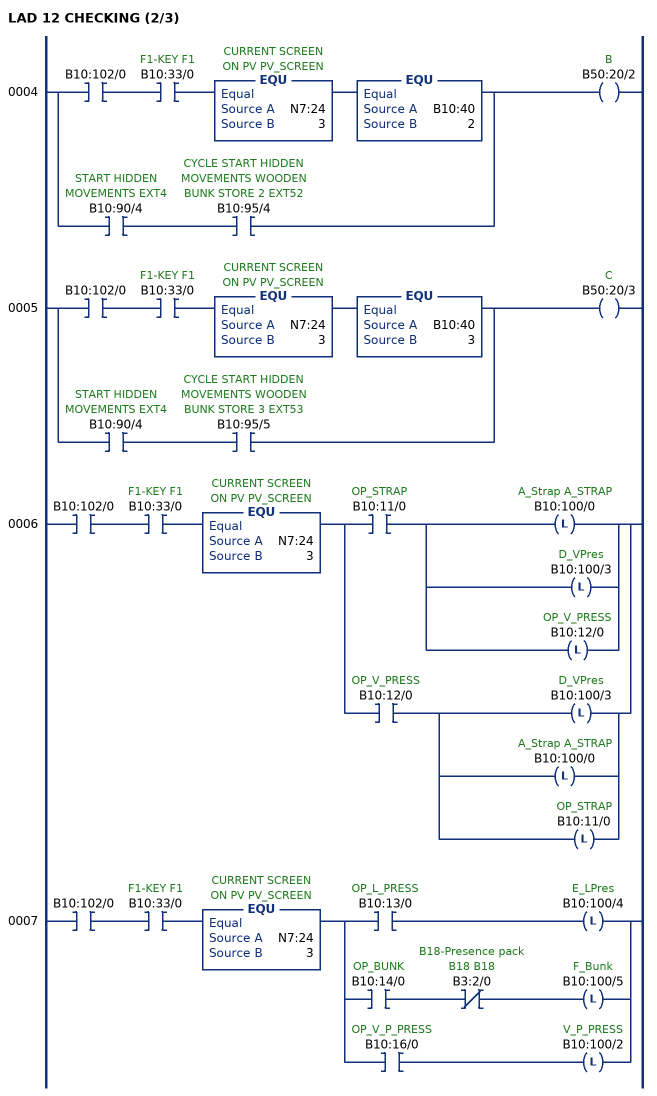
% Rung: 4 %
SOR BST XIC B10:102/0 XIC B10:33/0 EQU N7:24 3 EQU B10:40 2 NXB XIC B10:90/4 XIC B10:95/4 BND OTE B50:20/2 EOR
%   B10:33/0  F1  "F1-KEY" %
%   N7:24  PV_SCREEN  "CURRENT SCREEN ON PV" %
%   B10:90/4  EXT4  "START HIDDEN MOVEMENTS" %
%   B10:95/4  EXT52  "CYCLE START HIDDEN MOVEMENTS WOODEN BUNK STORE 2" %
%   B50:20/2  "B" %
% Rung: 5 %
SOR BST XIC B10:102/0 XIC B10:33/0 EQU N7:24 3 EQU B10:40 3 NXB XIC B10:90/4 XIC B10:95/5 BND OTE B50:20/3 EOR
%   B10:33/0  F1  "F1-KEY" %
%   N7:24  PV_SCREEN  "CURRENT SCREEN ON PV" %
%   B10:90/4  EXT4  "START HIDDEN MOVEMENTS" %
%   B10:95/5  EXT53  "CYCLE START HIDDEN MOVEMENTS WOODEN BUNK STORE 3" %
%   B50:20/3  "C" %
% Rung: 6 %
SOR XIC B10:102/0 XIC B10:33/0 EQU N7:24 3 BST XIC B10:11/0 BST OTL B10:100/0 NXB BST OTL B10:100/3 NXB OTL B10:12/0 BND BND NXB XIC B10:12/0 BST OTL B10:100/3 NXB BST OTL B10:100/0 NXB OTL B10:11/0 BND BND BND EOR
%   B10:33/0  F1  "F1-KEY" %
%   N7:24  PV_SCREEN  "CURRENT SCREEN ON PV" %
%   B10:11/0  "OP_STRAP" %
%   B10:100/0  A_STRAP  "A_Strap" %
%   B10:100/3  "D_VPres" %
%   B10:12/0  "OP_V_PRESS" %
% Rung: 7 %
SOR XIC B10:102/0 XIC B10:33/0 EQU N7:24 3 BST XIC B10:13/0 OTL B10:100/4 NXB BST XIC B10:14/0 XIO B3:2/0 OTL B10:100/5 NXB XIC B10:16/0 OTL B10:100/2 BND BND EOR
%   B10:33/0  F1  "F1-KEY" %
%   N7:24  PV_SCREEN  "CURRENT SCREEN ON PV" %
%   B10:13/0  "OP_L_PRESS" %
%   B10:100/4  "E_LPres" %
%   B10:14/0  "OP_BUNK" %
%   B3:2/0  B18  "B18-Presence pack B18" %
%   B10:100/5  "F_Bunk" %
%   B10:16/0  "OP_V_P_PRESS" %
%   B10:100/2  "V_P_PRESS" %

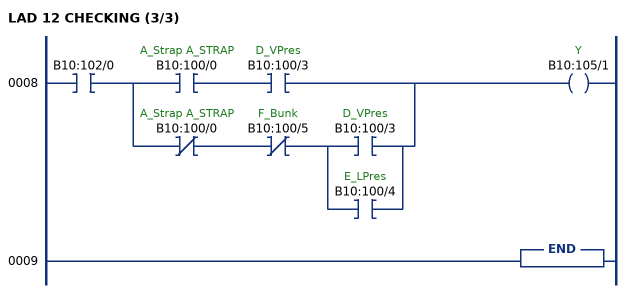
% Rung: 8 %
SOR XIC B10:102/0 BST XIC B10:100/0 XIC B10:100/3 NXB XIO B10:100/0 XIO B10:100/5 BST XIC B10:100/3 NXB XIC B10:100/4 BND BND OTE B10:105/1 EOR
%   B10:100/0  A_STRAP  "A_Strap" %
%   B10:100/3  "D_VPres" %
%   B10:100/5  "F_Bunk" %
%   B10:100/4  "E_LPres" %
%   B10:105/1  "Y" %
% Rung: 9 %
SOR END EOR

LADDER 13 "INFEED"    % INFEED CONTROLS %
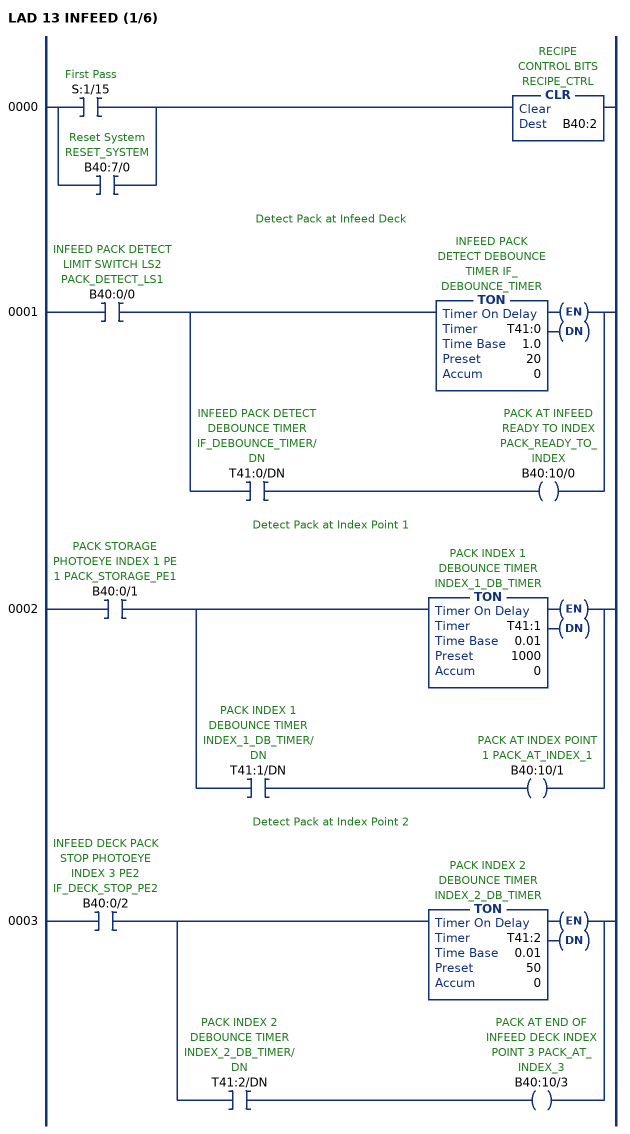
% Rung: 0 %
SOR BST XIC S:1/15 NXB XIC B40:7/0 BND CLR B40:2 EOR
%   S:1/15  "First Pass" %
%   B40:7/0  RESET_SYSTEM  "Reset System" %
%   B40:2  RECIPE_CTRL  "RECIPE CONTROL BITS" %
% Rung: 1 %
% Detect Pack at Infeed Deck %
SOR XIC B40:0/0 BST TON T41:0 1.0 20 0 NXB XIC T41:0/DN OTE B40:10/0 BND EOR
%   B40:0/0  PACK_DETECT_LS1  "INFEED PACK DETECT LIMIT SWITCH LS2" %
%   T41:0  IF_DEBOUNCE_TIMER  "INFEED PACK DETECT DEBOUNCE TIMER" %
%   B40:10/0  PACK_READY_TO_INDEX  "PACK AT INFEED READY TO INDEX" %
% Rung: 2 %
% Detect Pack at Index Point 1 %
SOR XIC B40:0/1 BST TON T41:1 0.01 1000 0 NXB XIC T41:1/DN OTE B40:10/1 BND EOR
%   B40:0/1  PACK_STORAGE_PE1  "PACK STORAGE PHOTOEYE INDEX 1 PE 1" %
%   T41:1  INDEX_1_DB_TIMER  "PACK INDEX 1 DEBOUNCE TIMER" %
%   B40:10/1  PACK_AT_INDEX_1  "PACK AT INDEX POINT 1" %
% Rung: 3 %
% Detect Pack at Index Point 2 %
SOR XIC B40:0/2 BST TON T41:2 0.01 50 0 NXB XIC T41:2/DN OTE B40:10/3 BND EOR
%   B40:0/2  IF_DECK_STOP_PE2  "INFEED DECK PACK STOP PHOTOEYE INDEX 3 PE2" %
%   T41:2  INDEX_2_DB_TIMER  "PACK INDEX 2 DEBOUNCE TIMER" %
%   B40:10/3  PACK_AT_INDEX_3  "PACK AT END OF INFEED DECK INDEX POINT 3" %

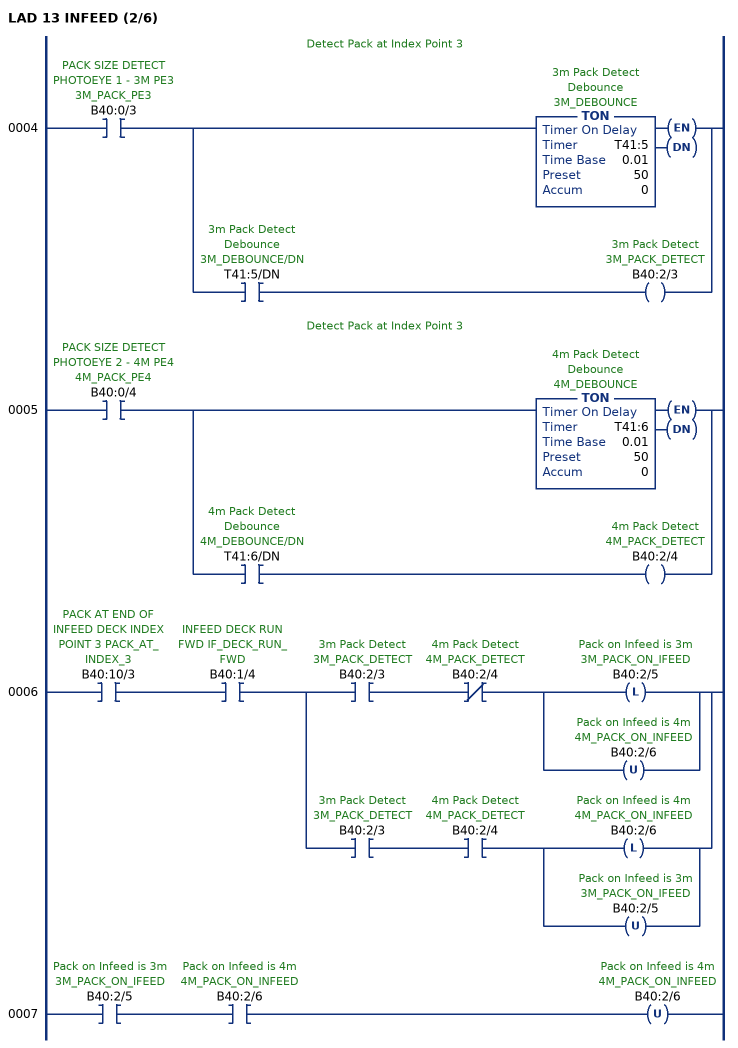
% Rung: 4 %
% Detect Pack at Index Point 3 %
SOR XIC B40:0/3 BST TON T41:5 0.01 50 0 NXB XIC T41:5/DN OTE B40:2/3 BND EOR
%   B40:0/3  3M_PACK_PE3  "PACK SIZE DETECT PHOTOEYE 1 - 3M PE3" %
%   T41:5  3M_DEBOUNCE  "3m Pack Detect Debounce" %
%   B40:2/3  3M_PACK_DETECT  "3m Pack Detect" %
% Rung: 5 %
% Detect Pack at Index Point 3 %
SOR XIC B40:0/4 BST TON T41:6 0.01 50 0 NXB XIC T41:6/DN OTE B40:2/4 BND EOR
%   B40:0/4  4M_PACK_PE4  "PACK SIZE DETECT PHOTOEYE 2 - 4M PE4" %
%   T41:6  4M_DEBOUNCE  "4m Pack Detect Debounce" %
%   B40:2/4  4M_PACK_DETECT  "4m Pack Detect" %
% Rung: 6 %
SOR XIC B40:10/3 XIC B40:1/4 BST XIC B40:2/3 XIO B40:2/4 BST OTL B40:2/5 NXB OTU B40:2/6 BND NXB XIC B40:2/3 XIC B40:2/4 BST OTL B40:2/6 NXB OTU B40:2/5 BND BND EOR
%   B40:10/3  PACK_AT_INDEX_3  "PACK AT END OF INFEED DECK INDEX POINT 3" %
%   B40:1/4  IF_DECK_RUN_FWD  "INFEED DECK RUN FWD" %
%   B40:2/3  3M_PACK_DETECT  "3m Pack Detect" %
%   B40:2/4  4M_PACK_DETECT  "4m Pack Detect" %
%   B40:2/5  3M_PACK_ON_IFEED  "Pack on Infeed is 3m" %
%   B40:2/6  4M_PACK_ON_INFEED  "Pack on Infeed is 4m" %
% Rung: 7 %
SOR XIC B40:2/5 XIC B40:2/6 OTU B40:2/6 EOR
%   B40:2/5  3M_PACK_ON_IFEED  "Pack on Infeed is 3m" %
%   B40:2/6  4M_PACK_ON_INFEED  "Pack on Infeed is 4m" %

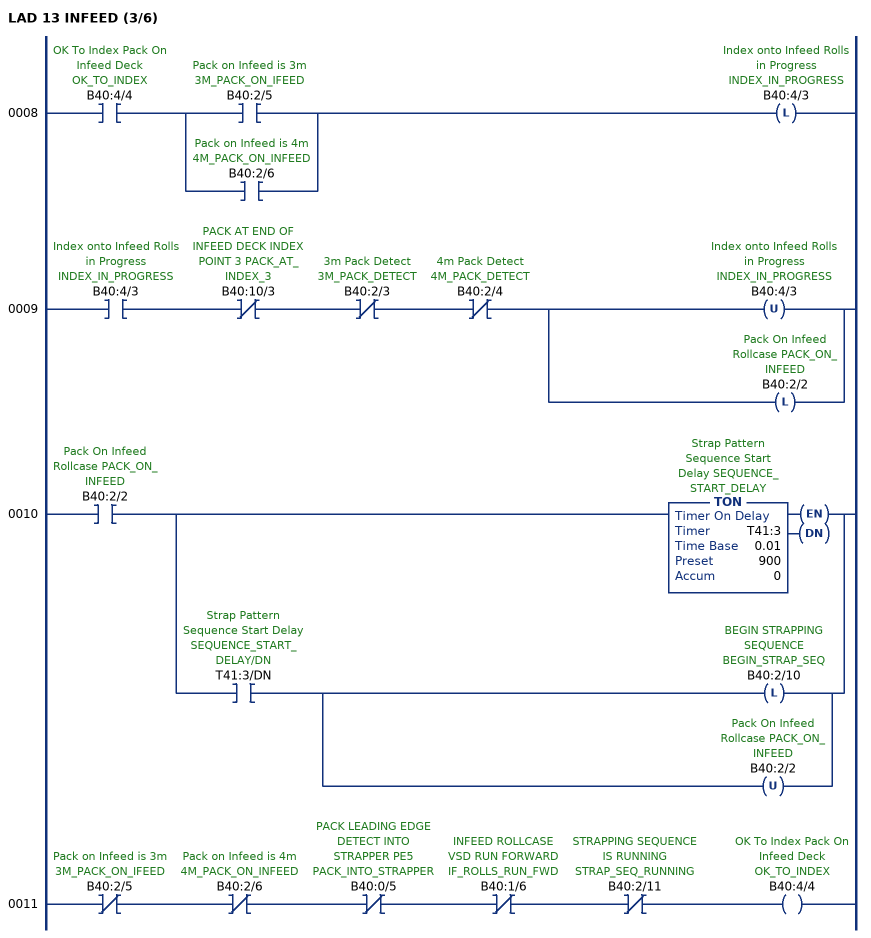
% Rung: 8 %
SOR XIC B40:4/4 BST XIC B40:2/5 NXB XIC B40:2/6 BND OTL B40:4/3 EOR
%   B40:4/4  OK_TO_INDEX  "OK To Index Pack On Infeed Deck" %
%   B40:2/5  3M_PACK_ON_IFEED  "Pack on Infeed is 3m" %
%   B40:2/6  4M_PACK_ON_INFEED  "Pack on Infeed is 4m" %
%   B40:4/3  INDEX_IN_PROGRESS  "Index onto Infeed Rolls in Progress" %
% Rung: 9 %
SOR XIC B40:4/3 XIO B40:10/3 XIO B40:2/3 XIO B40:2/4 BST OTU B40:4/3 NXB OTL B40:2/2 BND EOR
%   B40:4/3  INDEX_IN_PROGRESS  "Index onto Infeed Rolls in Progress" %
%   B40:10/3  PACK_AT_INDEX_3  "PACK AT END OF INFEED DECK INDEX POINT 3" %
%   B40:2/3  3M_PACK_DETECT  "3m Pack Detect" %
%   B40:2/4  4M_PACK_DETECT  "4m Pack Detect" %
%   B40:2/2  PACK_ON_INFEED  "Pack On Infeed Rollcase" %
% Rung: 10 %
SOR XIC B40:2/2 BST TON T41:3 0.01 900 0 NXB XIC T41:3/DN BST OTL B40:2/10 NXB OTU B40:2/2 BND BND EOR
%   B40:2/2  PACK_ON_INFEED  "Pack On Infeed Rollcase" %
%   T41:3  SEQUENCE_START_DELAY  "Strap Pattern Sequence Start Delay" %
%   B40:2/10  BEGIN_STRAP_SEQ  "BEGIN STRAPPING SEQUENCE" %
% Rung: 11 %
SOR XIO B40:2/5 XIO B40:2/6 XIO B40:0/5 XIO B40:1/6 XIO B40:2/11 OTE B40:4/4 EOR
%   B40:2/5  3M_PACK_ON_IFEED  "Pack on Infeed is 3m" %
%   B40:2/6  4M_PACK_ON_INFEED  "Pack on Infeed is 4m" %
%   B40:0/5  PACK_INTO_STRAPPER  "PACK LEADING EDGE DETECT INTO STRAPPER PE5" %
%   B40:1/6  IF_ROLLS_RUN_FWD  "INFEED ROLLCASE VSD RUN FORWARD" %
%   B40:2/11  STRAP_SEQ_RUNNING  "STRAPPING SEQUENCE IS RUNNING" %
%   B40:4/4  OK_TO_INDEX  "OK To Index Pack On Infeed Deck" %

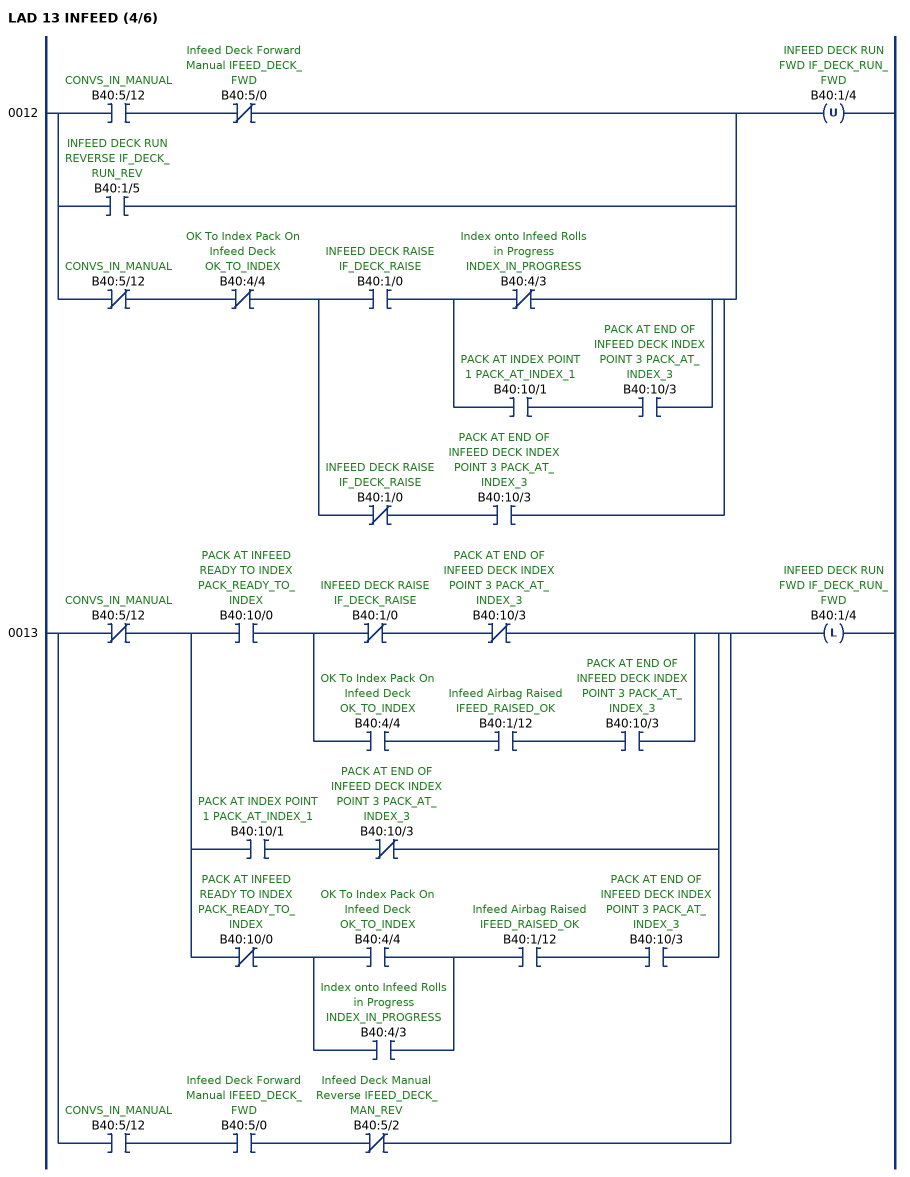
% Rung: 12 %
SOR BST XIC B40:5/12 XIO B40:5/0 NXB XIC B40:1/5 NXB XIO B40:5/12 XIO B40:4/4 BST XIC B40:1/0 BST XIO B40:4/3 NXB XIC B40:10/1 XIC B40:10/3 BND NXB XIO B40:1/0 XIC B40:10/3 BND BND OTU B40:1/4 EOR
%   B40:5/12  CONVS_IN_MANUAL %
%   B40:5/0  IFEED_DECK_FWD  "Infeed Deck Forward Manual" %
%   B40:1/5  IF_DECK_RUN_REV  "INFEED DECK RUN REVERSE" %
%   B40:4/4  OK_TO_INDEX  "OK To Index Pack On Infeed Deck" %
%   B40:1/0  IF_DECK_RAISE  "INFEED DECK RAISE" %
%   B40:4/3  INDEX_IN_PROGRESS  "Index onto Infeed Rolls in Progress" %
%   B40:10/1  PACK_AT_INDEX_1  "PACK AT INDEX POINT 1" %
%   B40:10/3  PACK_AT_INDEX_3  "PACK AT END OF INFEED DECK INDEX POINT 3" %
%   B40:1/4  IF_DECK_RUN_FWD  "INFEED DECK RUN FWD" %
% Rung: 13 %
SOR BST XIO B40:5/12 BST XIC B40:10/0 BST XIO B40:1/0 XIO B40:10/3 NXB XIC B40:4/4 XIC B40:1/12 XIC B40:10/3 BND NXB XIC B40:10/1 XIO B40:10/3 NXB XIO B40:10/0 BST XIC B40:4/4 NXB XIC B40:4/3 BND XIC B40:1/12 XIC B40:10/3 BND NXB XIC B40:5/12 XIC B40:5/0 XIO B40:5/2 BND OTL B40:1/4 EOR
%   B40:5/12  CONVS_IN_MANUAL %
%   B40:10/0  PACK_READY_TO_INDEX  "PACK AT INFEED READY TO INDEX" %
%   B40:1/0  IF_DECK_RAISE  "INFEED DECK RAISE" %
%   B40:10/3  PACK_AT_INDEX_3  "PACK AT END OF INFEED DECK INDEX POINT 3" %
%   B40:4/4  OK_TO_INDEX  "OK To Index Pack On Infeed Deck" %
%   B40:1/12  IFEED_RAISED_OK  "Infeed Airbag Raised" %
%   B40:10/1  PACK_AT_INDEX_1  "PACK AT INDEX POINT 1" %
%   B40:4/3  INDEX_IN_PROGRESS  "Index onto Infeed Rolls in Progress" %
%   B40:5/0  IFEED_DECK_FWD  "Infeed Deck Forward Manual" %
%   B40:5/2  IFEED_DECK_MAN_REV  "Infeed Deck Manual Reverse" %
%   B40:1/4  IF_DECK_RUN_FWD  "INFEED DECK RUN FWD" %

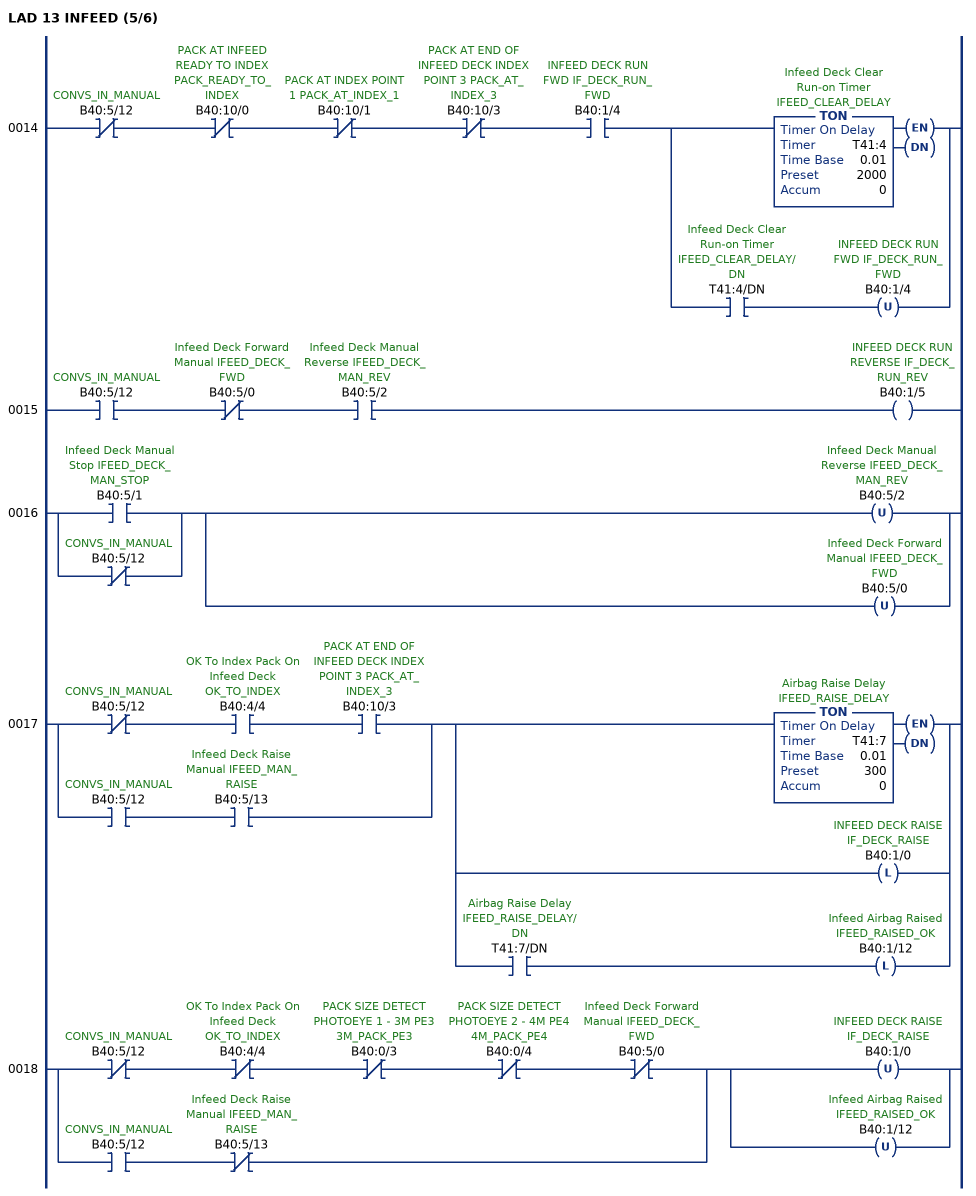
% Rung: 14 %
SOR XIO B40:5/12 XIO B40:10/0 XIO B40:10/1 XIO B40:10/3 XIC B40:1/4 BST TON T41:4 0.01 2000 0 NXB XIC T41:4/DN OTU B40:1/4 BND EOR
%   B40:5/12  CONVS_IN_MANUAL %
%   B40:10/0  PACK_READY_TO_INDEX  "PACK AT INFEED READY TO INDEX" %
%   B40:10/1  PACK_AT_INDEX_1  "PACK AT INDEX POINT 1" %
%   B40:10/3  PACK_AT_INDEX_3  "PACK AT END OF INFEED DECK INDEX POINT 3" %
%   B40:1/4  IF_DECK_RUN_FWD  "INFEED DECK RUN FWD" %
%   T41:4  IFEED_CLEAR_DELAY  "Infeed Deck Clear Run-on Timer" %
% Rung: 15 %
SOR XIC B40:5/12 XIO B40:5/0 XIC B40:5/2 OTE B40:1/5 EOR
%   B40:5/12  CONVS_IN_MANUAL %
%   B40:5/0  IFEED_DECK_FWD  "Infeed Deck Forward Manual" %
%   B40:5/2  IFEED_DECK_MAN_REV  "Infeed Deck Manual Reverse" %
%   B40:1/5  IF_DECK_RUN_REV  "INFEED DECK RUN REVERSE" %
% Rung: 16 %
SOR BST XIC B40:5/1 NXB XIO B40:5/12 BND BST OTU B40:5/2 NXB OTU B40:5/0 BND EOR
%   B40:5/1  IFEED_DECK_MAN_STOP  "Infeed Deck Manual Stop" %
%   B40:5/12  CONVS_IN_MANUAL %
%   B40:5/2  IFEED_DECK_MAN_REV  "Infeed Deck Manual Reverse" %
%   B40:5/0  IFEED_DECK_FWD  "Infeed Deck Forward Manual" %
% Rung: 17 %
SOR BST XIO B40:5/12 XIC B40:4/4 XIC B40:10/3 NXB XIC B40:5/12 XIC B40:5/13 BND BST TON T41:7 0.01 300 0 NXB OTL B40:1/0 NXB XIC T41:7/DN OTL B40:1/12 BND EOR
%   B40:5/12  CONVS_IN_MANUAL %
%   B40:4/4  OK_TO_INDEX  "OK To Index Pack On Infeed Deck" %
%   B40:10/3  PACK_AT_INDEX_3  "PACK AT END OF INFEED DECK INDEX POINT 3" %
%   B40:5/13  IFEED_MAN_RAISE  "Infeed Deck Raise Manual" %
%   T41:7  IFEED_RAISE_DELAY  "Airbag Raise Delay" %
%   B40:1/0  IF_DECK_RAISE  "INFEED DECK RAISE" %
%   B40:1/12  IFEED_RAISED_OK  "Infeed Airbag Raised" %
% Rung: 18 %
SOR BST XIO B40:5/12 XIO B40:4/4 XIO B40:0/3 XIO B40:0/4 XIO B40:5/0 NXB XIC B40:5/12 XIO B40:5/13 BND BST OTU B40:1/0 NXB OTU B40:1/12 BND EOR
%   B40:5/12  CONVS_IN_MANUAL %
%   B40:4/4  OK_TO_INDEX  "OK To Index Pack On Infeed Deck" %
%   B40:0/3  3M_PACK_PE3  "PACK SIZE DETECT PHOTOEYE 1 - 3M PE3" %
%   B40:0/4  4M_PACK_PE4  "PACK SIZE DETECT PHOTOEYE 2 - 4M PE4" %
%   B40:5/0  IFEED_DECK_FWD  "Infeed Deck Forward Manual" %
%   B40:5/13  IFEED_MAN_RAISE  "Infeed Deck Raise Manual" %
%   B40:1/0  IF_DECK_RAISE  "INFEED DECK RAISE" %
%   B40:1/12  IFEED_RAISED_OK  "Infeed Airbag Raised" %

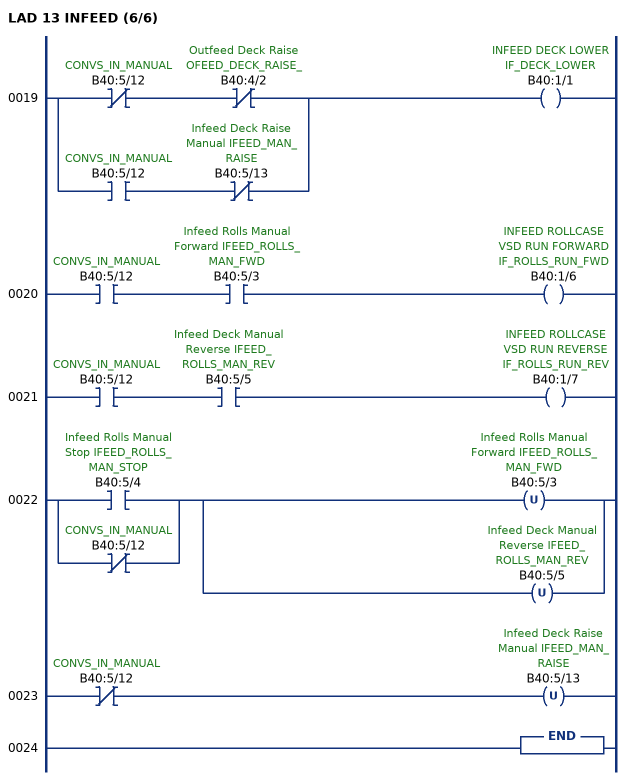
% Rung: 19 %
SOR BST XIO B40:5/12 XIO B40:4/2 NXB XIC B40:5/12 XIO B40:5/13 BND OTE B40:1/1 EOR
%   B40:5/12  CONVS_IN_MANUAL %
%   B40:4/2  OFEED_DECK_RAISE_  "Outfeed Deck Raise" %
%   B40:5/13  IFEED_MAN_RAISE  "Infeed Deck Raise Manual" %
%   B40:1/1  IF_DECK_LOWER  "INFEED DECK LOWER" %
% Rung: 20 %
SOR XIC B40:5/12 XIC B40:5/3 OTE B40:1/6 EOR
%   B40:5/12  CONVS_IN_MANUAL %
%   B40:5/3  IFEED_ROLLS_MAN_FWD  "Infeed Rolls Manual Forward" %
%   B40:1/6  IF_ROLLS_RUN_FWD  "INFEED ROLLCASE VSD RUN FORWARD" %
% Rung: 21 %
SOR XIC B40:5/12 XIC B40:5/5 OTE B40:1/7 EOR
%   B40:5/12  CONVS_IN_MANUAL %
%   B40:5/5  IFEED_ROLLS_MAN_REV  "Infeed Deck Manual Reverse" %
%   B40:1/7  IF_ROLLS_RUN_REV  "INFEED ROLLCASE VSD RUN REVERSE" %
% Rung: 22 %
SOR BST XIC B40:5/4 NXB XIO B40:5/12 BND BST OTU B40:5/3 NXB OTU B40:5/5 BND EOR
%   B40:5/4  IFEED_ROLLS_MAN_STOP  "Infeed Rolls Manual Stop" %
%   B40:5/12  CONVS_IN_MANUAL %
%   B40:5/3  IFEED_ROLLS_MAN_FWD  "Infeed Rolls Manual Forward" %
%   B40:5/5  IFEED_ROLLS_MAN_REV  "Infeed Deck Manual Reverse" %
% Rung: 23 %
SOR XIO B40:5/12 OTU B40:5/13 EOR
%   B40:5/12  CONVS_IN_MANUAL %
%   B40:5/13  IFEED_MAN_RAISE  "Infeed Deck Raise Manual" %
% Rung: 24 %
SOR END EOR

LADDER 14 "OUTFEED"    % OUTFEED CONTROLS %
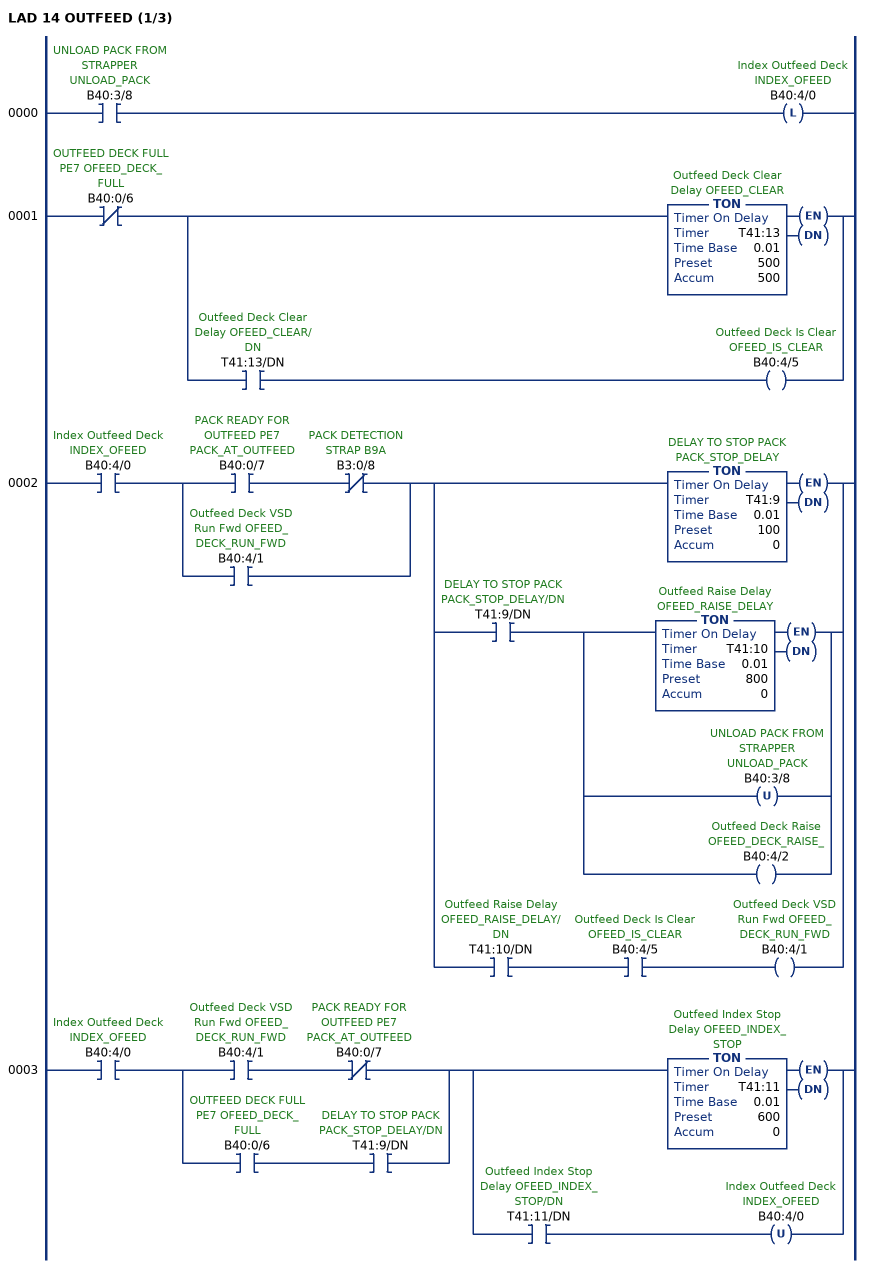
% Rung: 0 %
SOR XIC B40:3/8 OTL B40:4/0 EOR
%   B40:3/8  UNLOAD_PACK  "UNLOAD PACK FROM STRAPPER" %
%   B40:4/0  INDEX_OFEED  "Index Outfeed Deck" %
% Rung: 1 %
SOR XIO B40:0/6 BST TON T41:13 0.01 500 500 NXB XIC T41:13/DN OTE B40:4/5 BND EOR
%   B40:0/6  OFEED_DECK_FULL  "OUTFEED DECK FULL PE7" %
%   T41:13  OFEED_CLEAR  "Outfeed Deck Clear Delay" %
%   B40:4/5  OFEED_IS_CLEAR  "Outfeed Deck Is Clear" %
% Rung: 2 %
SOR XIC B40:4/0 BST XIC B40:0/7 XIO B3:0/8 NXB XIC B40:4/1 BND BST TON T41:9 0.01 100 0 NXB XIC T41:9/DN BST TON T41:10 0.01 800 0 NXB OTU B40:3/8 NXB OTE B40:4/2 BND NXB XIC T41:10/DN XIC B40:4/5 OTE B40:4/1 BND EOR
%   B40:4/0  INDEX_OFEED  "Index Outfeed Deck" %
%   B40:0/7  PACK_AT_OUTFEED  "PACK READY FOR OUTFEED PE7" %
%   B3:0/8  B9A  "PACK DETECTION STRAP" %
%   B40:4/1  OFEED_DECK_RUN_FWD  "Outfeed Deck VSD Run Fwd" %
%   T41:9  PACK_STOP_DELAY  "DELAY TO STOP PACK" %
%   T41:10  OFEED_RAISE_DELAY  "Outfeed Raise Delay" %
%   B40:3/8  UNLOAD_PACK  "UNLOAD PACK FROM STRAPPER" %
%   B40:4/2  OFEED_DECK_RAISE_  "Outfeed Deck Raise" %
%   B40:4/5  OFEED_IS_CLEAR  "Outfeed Deck Is Clear" %
% Rung: 3 %
SOR XIC B40:4/0 BST XIC B40:4/1 XIO B40:0/7 NXB XIC B40:0/6 XIC T41:9/DN BND BST TON T41:11 0.01 600 0 NXB XIC T41:11/DN OTU B40:4/0 BND EOR
%   B40:4/0  INDEX_OFEED  "Index Outfeed Deck" %
%   B40:4/1  OFEED_DECK_RUN_FWD  "Outfeed Deck VSD Run Fwd" %
%   B40:0/7  PACK_AT_OUTFEED  "PACK READY FOR OUTFEED PE7" %
%   B40:0/6  OFEED_DECK_FULL  "OUTFEED DECK FULL PE7" %
%   T41:9  PACK_STOP_DELAY  "DELAY TO STOP PACK" %
%   T41:11  OFEED_INDEX_STOP  "Outfeed Index Stop Delay" %

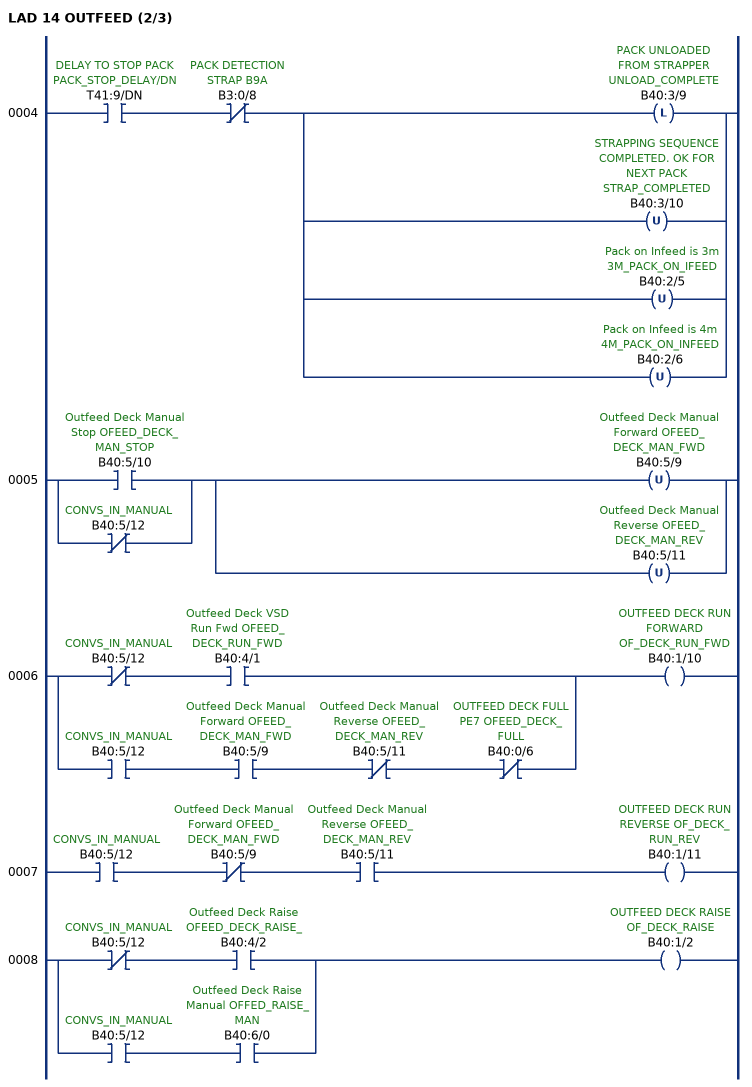
% Rung: 4 %
SOR XIC T41:9/DN XIO B3:0/8 BST OTL B40:3/9 NXB OTU B40:3/10 NXB OTU B40:2/5 NXB OTU B40:2/6 BND EOR
%   T41:9  PACK_STOP_DELAY  "DELAY TO STOP PACK" %
%   B3:0/8  B9A  "PACK DETECTION STRAP" %
%   B40:3/9  UNLOAD_COMPLETE  "PACK UNLOADED FROM STRAPPER" %
%   B40:3/10  STRAP_COMPLETED  "STRAPPING SEQUENCE COMPLETED. OK FOR NEXT PACK" %
%   B40:2/5  3M_PACK_ON_IFEED  "Pack on Infeed is 3m" %
%   B40:2/6  4M_PACK_ON_INFEED  "Pack on Infeed is 4m" %
% Rung: 5 %
SOR BST XIC B40:5/10 NXB XIO B40:5/12 BND BST OTU B40:5/9 NXB OTU B40:5/11 BND EOR
%   B40:5/10  OFEED_DECK_MAN_STOP  "Outfeed Deck Manual Stop" %
%   B40:5/12  CONVS_IN_MANUAL %
%   B40:5/9  OFEED_DECK_MAN_FWD  "Outfeed Deck Manual Forward" %
%   B40:5/11  OFEED_DECK_MAN_REV  "Outfeed Deck Manual Reverse" %
% Rung: 6 %
SOR BST XIO B40:5/12 XIC B40:4/1 NXB XIC B40:5/12 XIC B40:5/9 XIO B40:5/11 XIO B40:0/6 BND OTE B40:1/10 EOR
%   B40:5/12  CONVS_IN_MANUAL %
%   B40:4/1  OFEED_DECK_RUN_FWD  "Outfeed Deck VSD Run Fwd" %
%   B40:5/9  OFEED_DECK_MAN_FWD  "Outfeed Deck Manual Forward" %
%   B40:5/11  OFEED_DECK_MAN_REV  "Outfeed Deck Manual Reverse" %
%   B40:0/6  OFEED_DECK_FULL  "OUTFEED DECK FULL PE7" %
%   B40:1/10  OF_DECK_RUN_FWD  "OUTFEED DECK RUN FORWARD" %
% Rung: 7 %
SOR XIC B40:5/12 XIO B40:5/9 XIC B40:5/11 OTE B40:1/11 EOR
%   B40:5/12  CONVS_IN_MANUAL %
%   B40:5/9  OFEED_DECK_MAN_FWD  "Outfeed Deck Manual Forward" %
%   B40:5/11  OFEED_DECK_MAN_REV  "Outfeed Deck Manual Reverse" %
%   B40:1/11  OF_DECK_RUN_REV  "OUTFEED DECK RUN REVERSE" %
% Rung: 8 %
SOR BST XIO B40:5/12 XIC B40:4/2 NXB XIC B40:5/12 XIC B40:6/0 BND OTE B40:1/2 EOR
%   B40:5/12  CONVS_IN_MANUAL %
%   B40:4/2  OFEED_DECK_RAISE_  "Outfeed Deck Raise" %
%   B40:6/0  OFFED_RAISE_MAN  "Outfeed Deck Raise Manual" %
%   B40:1/2  OF_DECK_RAISE  "OUTFEED DECK RAISE" %

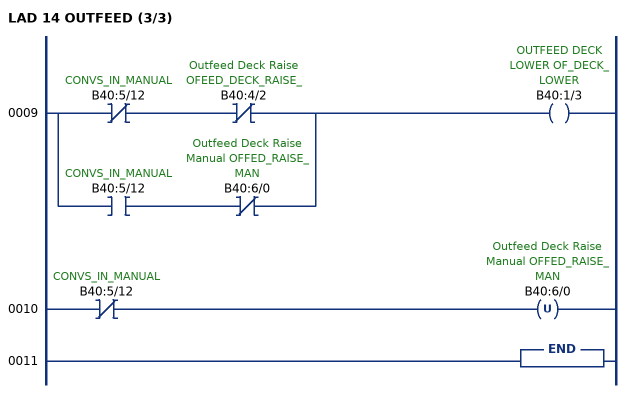
% Rung: 9 %
SOR BST XIO B40:5/12 XIO B40:4/2 NXB XIC B40:5/12 XIO B40:6/0 BND OTE B40:1/3 EOR
%   B40:5/12  CONVS_IN_MANUAL %
%   B40:4/2  OFEED_DECK_RAISE_  "Outfeed Deck Raise" %
%   B40:6/0  OFFED_RAISE_MAN  "Outfeed Deck Raise Manual" %
%   B40:1/3  OF_DECK_LOWER  "OUTFEED DECK LOWER" %
% Rung: 10 %
SOR XIO B40:5/12 OTU B40:6/0 EOR
%   B40:5/12  CONVS_IN_MANUAL %
%   B40:6/0  OFFED_RAISE_MAN  "Outfeed Deck Raise Manual" %
% Rung: 11 %
SOR END EOR

LADDER 15 "RECIPES"    % PV RECIPE CONTROL %
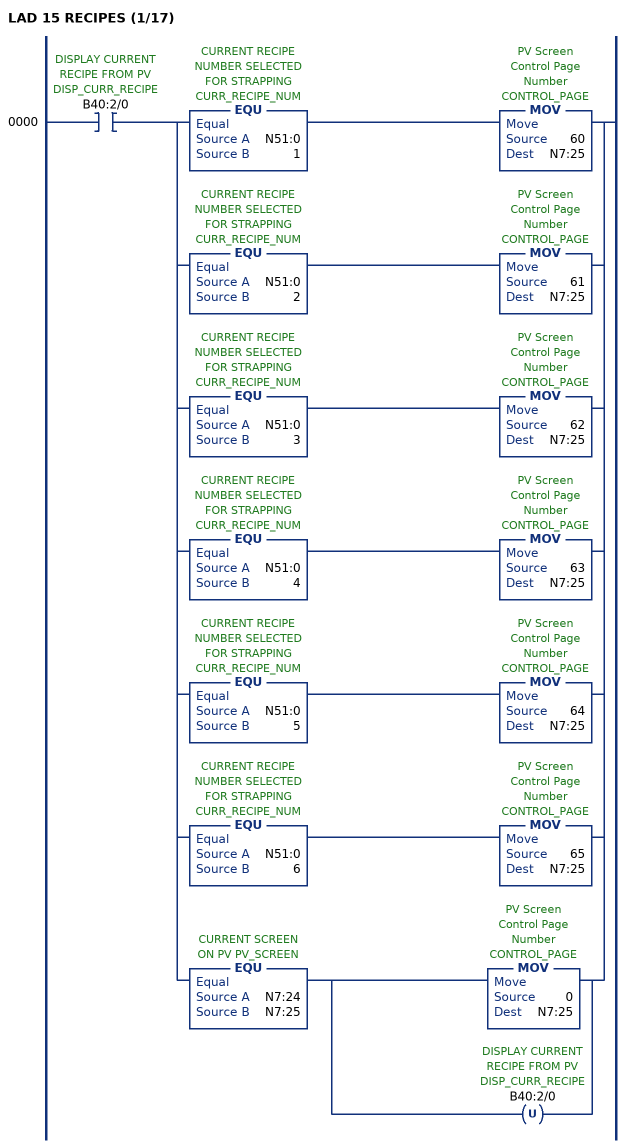
% Rung: 0 %
SOR XIC B40:2/0 BST EQU N51:0 1 MOV 60 N7:25 NXB EQU N51:0 2 MOV 61 N7:25 NXB EQU N51:0 3 MOV 62 N7:25 NXB EQU N51:0 4 MOV 63 N7:25 NXB EQU N51:0 5 MOV 64 N7:25 NXB EQU N51:0 6 MOV 65 N7:25 NXB EQU N7:24 N7:25 BST MOV 0 N7:25 NXB OTU B40:2/0 BND BND EOR
%   B40:2/0  DISP_CURR_RECIPE  "DISPLAY CURRENT RECIPE FROM PV" %
%   N51:0  CURR_RECIPE_NUM  "CURRENT RECIPE NUMBER SELECTED FOR STRAPPING" %
%   N7:25  CONTROL_PAGE  "PV Screen Control Page Number" %
%   N7:24  PV_SCREEN  "CURRENT SCREEN ON PV" %

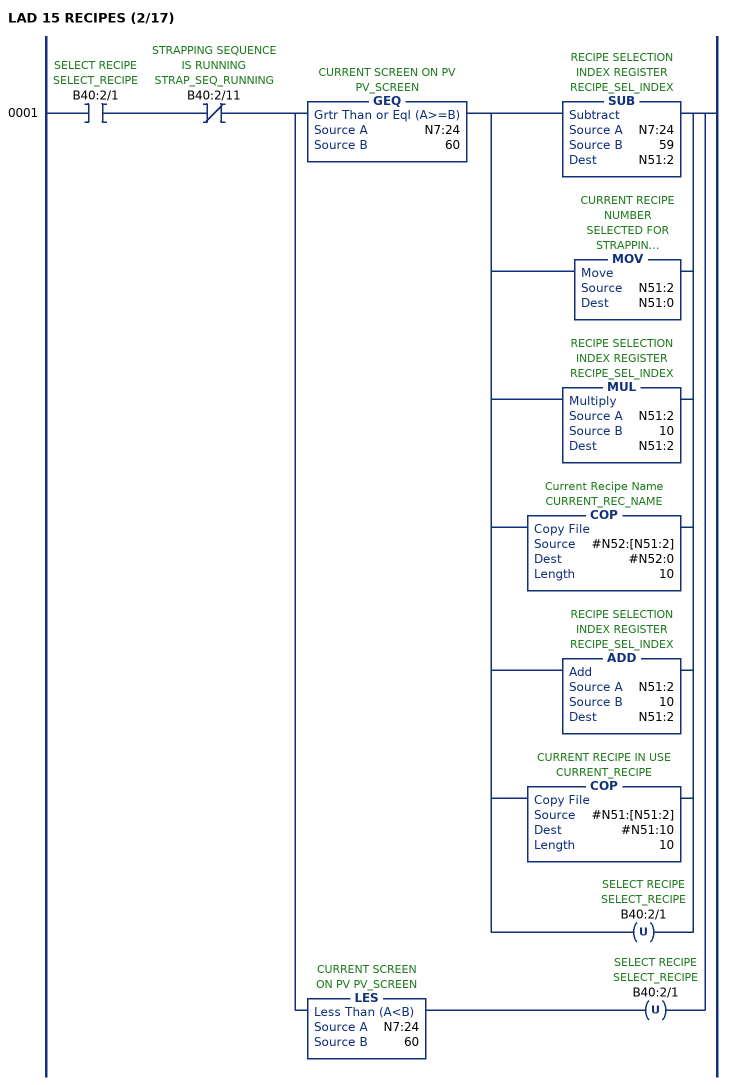
% Rung: 1 %
SOR XIC B40:2/1 XIO B40:2/11 BST GEQ N7:24 60 BST SUB N7:24 59 N51:2 NXB MOV N51:2 N51:0 NXB MUL N51:2 10 N51:2 NXB COP #N52:[N51:2] #N52:0 10 NXB ADD N51:2 10 N51:2 NXB COP #N51:[N51:2] #N51:10 10 NXB OTU B40:2/1 BND NXB LES N7:24 60 OTU B40:2/1 BND EOR
%   B40:2/1  SELECT_RECIPE  "SELECT RECIPE" %
%   B40:2/11  STRAP_SEQ_RUNNING  "STRAPPING SEQUENCE IS RUNNING" %
%   N7:24  PV_SCREEN  "CURRENT SCREEN ON PV" %
%   N51:2  RECIPE_SEL_INDEX  "RECIPE SELECTION INDEX REGISTER" %
%   N51:0  CURR_RECIPE_NUM  "CURRENT RECIPE NUMBER SELECTED FOR STRAPPING" %
%   N52:0  CURRENT_REC_NAME  "Current Recipe Name" %
%   N51:10  CURRENT_RECIPE  "CURRENT RECIPE IN USE" %

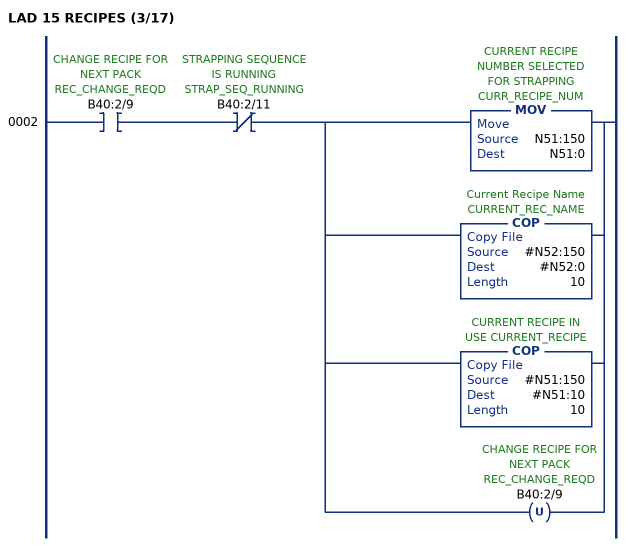
% Rung: 2 %
SOR XIC B40:2/9 XIO B40:2/11 BST MOV N51:150 N51:0 NXB COP #N52:150 #N52:0 10 NXB COP #N51:150 #N51:10 10 NXB OTU B40:2/9 BND EOR
%   B40:2/9  REC_CHANGE_REQD  "CHANGE RECIPE FOR NEXT PACK" %
%   B40:2/11  STRAP_SEQ_RUNNING  "STRAPPING SEQUENCE IS RUNNING" %
%   N51:150  RECIPE_14  "RECIPE 14" %
%   N51:0  CURR_RECIPE_NUM  "CURRENT RECIPE NUMBER SELECTED FOR STRAPPING" %
%   N52:0  CURRENT_REC_NAME  "Current Recipe Name" %
%   N51:10  CURRENT_RECIPE  "CURRENT RECIPE IN USE" %

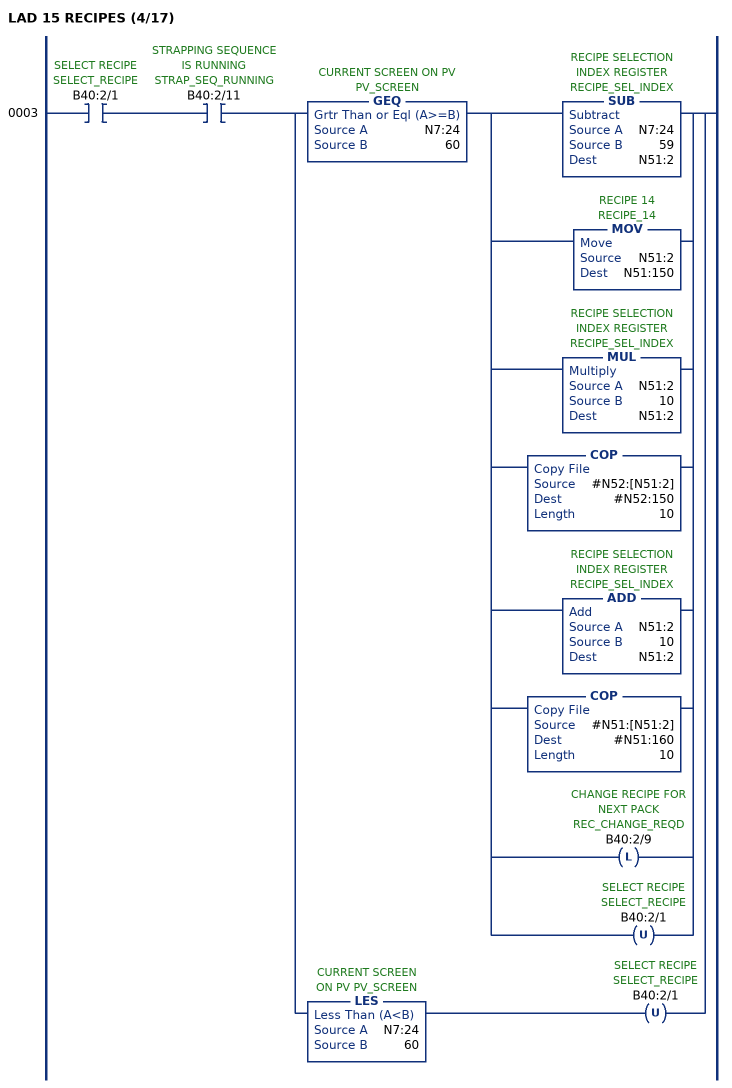
% Rung: 3 %
SOR XIC B40:2/1 XIC B40:2/11 BST GEQ N7:24 60 BST SUB N7:24 59 N51:2 NXB MOV N51:2 N51:150 NXB MUL N51:2 10 N51:2 NXB COP #N52:[N51:2] #N52:150 10 NXB ADD N51:2 10 N51:2 NXB COP #N51:[N51:2] #N51:160 10 NXB OTL B40:2/9 NXB OTU B40:2/1 BND NXB LES N7:24 60 OTU B40:2/1 BND EOR
%   B40:2/1  SELECT_RECIPE  "SELECT RECIPE" %
%   B40:2/11  STRAP_SEQ_RUNNING  "STRAPPING SEQUENCE IS RUNNING" %
%   N7:24  PV_SCREEN  "CURRENT SCREEN ON PV" %
%   N51:2  RECIPE_SEL_INDEX  "RECIPE SELECTION INDEX REGISTER" %
%   N51:150  RECIPE_14  "RECIPE 14" %
%   B40:2/9  REC_CHANGE_REQD  "CHANGE RECIPE FOR NEXT PACK" %

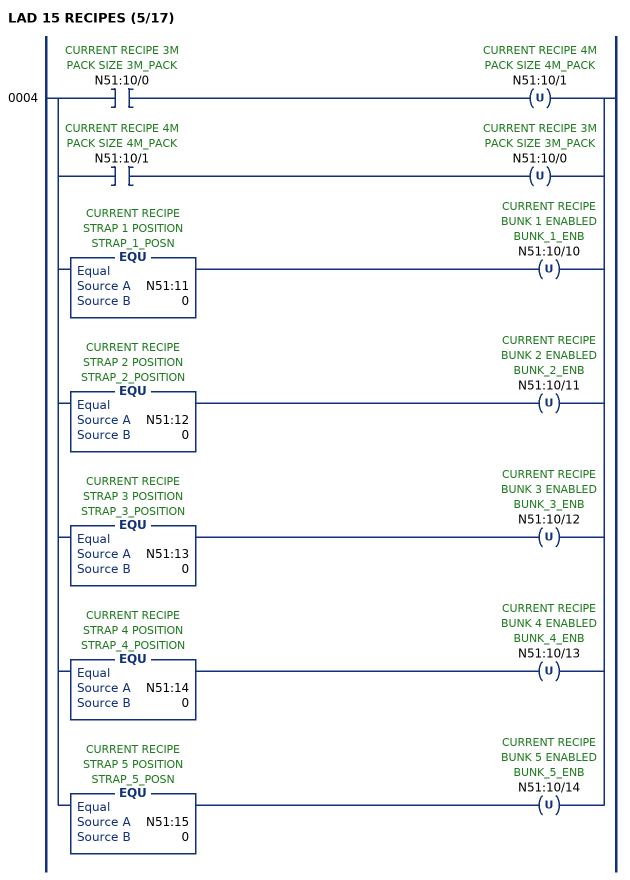
% Rung: 4 %
SOR BST XIC N51:10/0 OTU N51:10/1 NXB XIC N51:10/1 OTU N51:10/0 NXB EQU N51:11 0 OTU N51:10/10 NXB EQU N51:12 0 OTU N51:10/11 NXB EQU N51:13 0 OTU N51:10/12 NXB EQU N51:14 0 OTU N51:10/13 NXB EQU N51:15 0 OTU N51:10/14 BND EOR
%   N51:10/0  3M_PACK  "CURRENT RECIPE 3M PACK SIZE" %
%   N51:10/1  4M_PACK  "CURRENT RECIPE 4M PACK SIZE" %
%   N51:11  STRAP_1_POSN  "CURRENT RECIPE STRAP 1 POSITION" %
%   N51:10/10  BUNK_1_ENB  "CURRENT RECIPE BUNK 1 ENABLED" %
%   N51:12  STRAP_2_POSITION  "CURRENT RECIPE STRAP 2 POSITION" %
%   N51:10/11  BUNK_2_ENB  "CURRENT RECIPE BUNK 2 ENABLED" %
%   N51:13  STRAP_3_POSITION  "CURRENT RECIPE STRAP 3 POSITION" %
%   N51:10/12  BUNK_3_ENB  "CURRENT RECIPE BUNK 3 ENABLED" %
%   N51:14  STRAP_4_POSITION  "CURRENT RECIPE STRAP 4 POSITION" %
%   N51:10/13  BUNK_4_ENB  "CURRENT RECIPE BUNK 4 ENABLED" %
%   N51:15  STRAP_5_POSN  "CURRENT RECIPE STRAP 5 POSITION" %
%   N51:10/14  BUNK_5_ENB  "CURRENT RECIPE BUNK 5 ENABLED" %

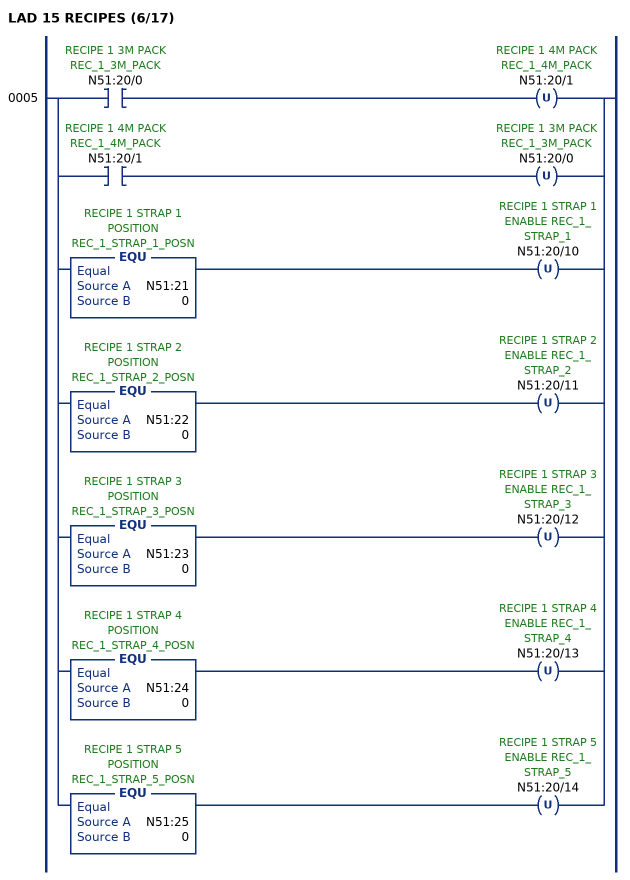
% Rung: 5 %
SOR BST XIC N51:20/0 OTU N51:20/1 NXB XIC N51:20/1 OTU N51:20/0 NXB EQU N51:21 0 OTU N51:20/10 NXB EQU N51:22 0 OTU N51:20/11 NXB EQU N51:23 0 OTU N51:20/12 NXB EQU N51:24 0 OTU N51:20/13 NXB EQU N51:25 0 OTU N51:20/14 BND EOR
%   N51:20/0  REC_1_3M_PACK  "RECIPE 1 3M PACK" %
%   N51:20/1  REC_1_4M_PACK  "RECIPE 1 4M PACK" %
%   N51:21  REC_1_STRAP_1_POSN  "RECIPE 1 STRAP 1 POSITION" %
%   N51:20/10  REC_1_STRAP_1  "RECIPE 1 STRAP 1 ENABLE" %
%   N51:22  REC_1_STRAP_2_POSN  "RECIPE 1 STRAP 2 POSITION" %
%   N51:20/11  REC_1_STRAP_2  "RECIPE 1 STRAP 2 ENABLE" %
%   N51:23  REC_1_STRAP_3_POSN  "RECIPE 1 STRAP 3 POSITION" %
%   N51:20/12  REC_1_STRAP_3  "RECIPE 1 STRAP 3 ENABLE" %
%   N51:24  REC_1_STRAP_4_POSN  "RECIPE 1 STRAP 4 POSITION" %
%   N51:20/13  REC_1_STRAP_4  "RECIPE 1 STRAP 4 ENABLE" %
%   N51:25  REC_1_STRAP_5_POSN  "RECIPE 1 STRAP 5 POSITION" %
%   N51:20/14  REC_1_STRAP_5  "RECIPE 1 STRAP 5 ENABLE" %

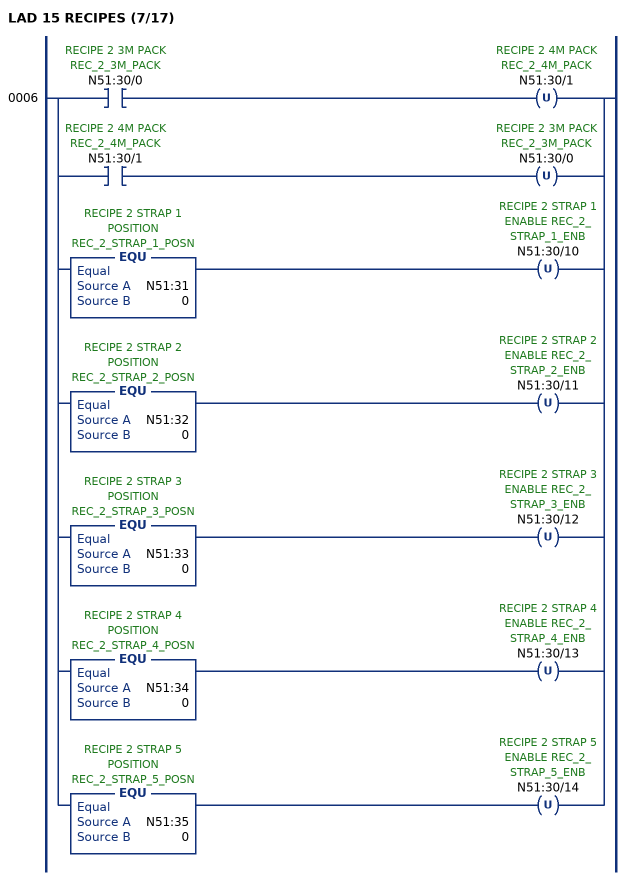
% Rung: 6 %
SOR BST XIC N51:30/0 OTU N51:30/1 NXB XIC N51:30/1 OTU N51:30/0 NXB EQU N51:31 0 OTU N51:30/10 NXB EQU N51:32 0 OTU N51:30/11 NXB EQU N51:33 0 OTU N51:30/12 NXB EQU N51:34 0 OTU N51:30/13 NXB EQU N51:35 0 OTU N51:30/14 BND EOR
%   N51:30/0  REC_2_3M_PACK  "RECIPE 2 3M PACK" %
%   N51:30/1  REC_2_4M_PACK  "RECIPE 2 4M PACK" %
%   N51:31  REC_2_STRAP_1_POSN  "RECIPE 2 STRAP 1 POSITION" %
%   N51:30/10  REC_2_STRAP_1_ENB  "RECIPE 2 STRAP 1 ENABLE" %
%   N51:32  REC_2_STRAP_2_POSN  "RECIPE 2 STRAP 2 POSITION" %
%   N51:30/11  REC_2_STRAP_2_ENB  "RECIPE 2 STRAP 2 ENABLE" %
%   N51:33  REC_2_STRAP_3_POSN  "RECIPE 2 STRAP 3 POSITION" %
%   N51:30/12  REC_2_STRAP_3_ENB  "RECIPE 2 STRAP 3 ENABLE" %
%   N51:34  REC_2_STRAP_4_POSN  "RECIPE 2 STRAP 4 POSITION" %
%   N51:30/13  REC_2_STRAP_4_ENB  "RECIPE 2 STRAP 4 ENABLE" %
%   N51:35  REC_2_STRAP_5_POSN  "RECIPE 2 STRAP 5 POSITION" %
%   N51:30/14  REC_2_STRAP_5_ENB  "RECIPE 2 STRAP 5 ENABLE" %

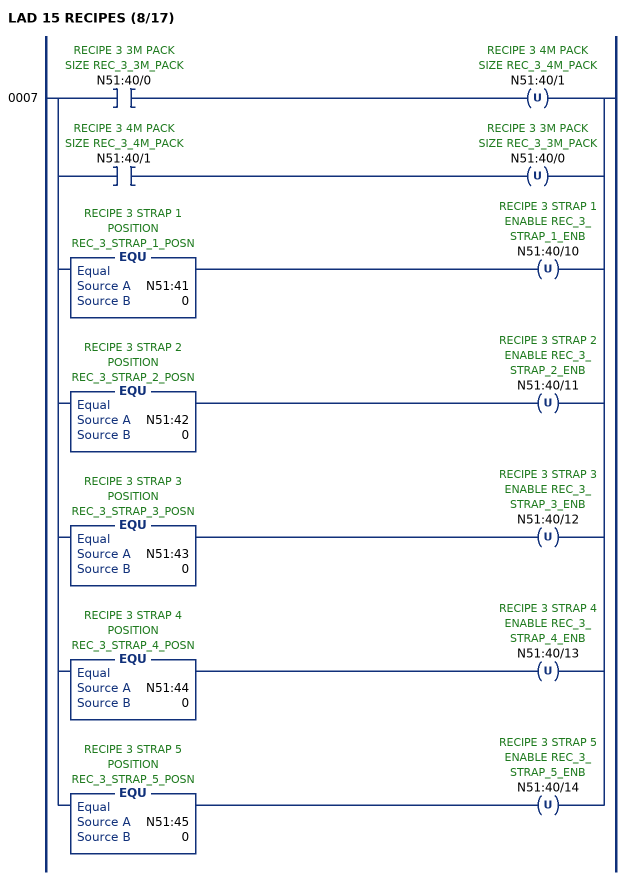
% Rung: 7 %
SOR BST XIC N51:40/0 OTU N51:40/1 NXB XIC N51:40/1 OTU N51:40/0 NXB EQU N51:41 0 OTU N51:40/10 NXB EQU N51:42 0 OTU N51:40/11 NXB EQU N51:43 0 OTU N51:40/12 NXB EQU N51:44 0 OTU N51:40/13 NXB EQU N51:45 0 OTU N51:40/14 BND EOR
%   N51:40/0  REC_3_3M_PACK  "RECIPE 3 3M PACK SIZE" %
%   N51:40/1  REC_3_4M_PACK  "RECIPE 3 4M PACK SIZE" %
%   N51:41  REC_3_STRAP_1_POSN  "RECIPE 3 STRAP 1 POSITION" %
%   N51:40/10  REC_3_STRAP_1_ENB  "RECIPE 3 STRAP 1 ENABLE" %
%   N51:42  REC_3_STRAP_2_POSN  "RECIPE 3 STRAP 2 POSITION" %
%   N51:40/11  REC_3_STRAP_2_ENB  "RECIPE 3 STRAP 2 ENABLE" %
%   N51:43  REC_3_STRAP_3_POSN  "RECIPE 3 STRAP 3 POSITION" %
%   N51:40/12  REC_3_STRAP_3_ENB  "RECIPE 3 STRAP 3 ENABLE" %
%   N51:44  REC_3_STRAP_4_POSN  "RECIPE 3 STRAP 4 POSITION" %
%   N51:40/13  REC_3_STRAP_4_ENB  "RECIPE 3 STRAP 4 ENABLE" %
%   N51:45  REC_3_STRAP_5_POSN  "RECIPE 3 STRAP 5 POSITION" %
%   N51:40/14  REC_3_STRAP_5_ENB  "RECIPE 3 STRAP 5 ENABLE" %

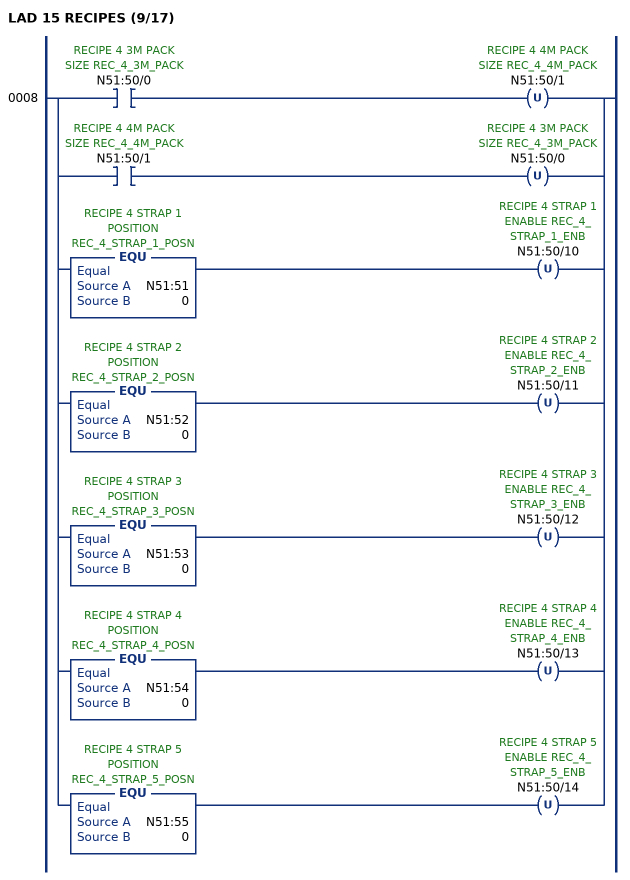
% Rung: 8 %
SOR BST XIC N51:50/0 OTU N51:50/1 NXB XIC N51:50/1 OTU N51:50/0 NXB EQU N51:51 0 OTU N51:50/10 NXB EQU N51:52 0 OTU N51:50/11 NXB EQU N51:53 0 OTU N51:50/12 NXB EQU N51:54 0 OTU N51:50/13 NXB EQU N51:55 0 OTU N51:50/14 BND EOR
%   N51:50/0  REC_4_3M_PACK  "RECIPE 4 3M PACK SIZE" %
%   N51:50/1  REC_4_4M_PACK  "RECIPE 4 4M PACK SIZE" %
%   N51:51  REC_4_STRAP_1_POSN  "RECIPE 4 STRAP 1 POSITION" %
%   N51:50/10  REC_4_STRAP_1_ENB  "RECIPE 4 STRAP 1 ENABLE" %
%   N51:52  REC_4_STRAP_2_POSN  "RECIPE 4 STRAP 2 POSITION" %
%   N51:50/11  REC_4_STRAP_2_ENB  "RECIPE 4 STRAP 2 ENABLE" %
%   N51:53  REC_4_STRAP_3_POSN  "RECIPE 4 STRAP 3 POSITION" %
%   N51:50/12  REC_4_STRAP_3_ENB  "RECIPE 4 STRAP 3 ENABLE" %
%   N51:54  REC_4_STRAP_4_POSN  "RECIPE 4 STRAP 4 POSITION" %
%   N51:50/13  REC_4_STRAP_4_ENB  "RECIPE 4 STRAP 4 ENABLE" %
%   N51:55  REC_4_STRAP_5_POSN  "RECIPE 4 STRAP 5 POSITION" %
%   N51:50/14  REC_4_STRAP_5_ENB  "RECIPE 4 STRAP 5 ENABLE" %

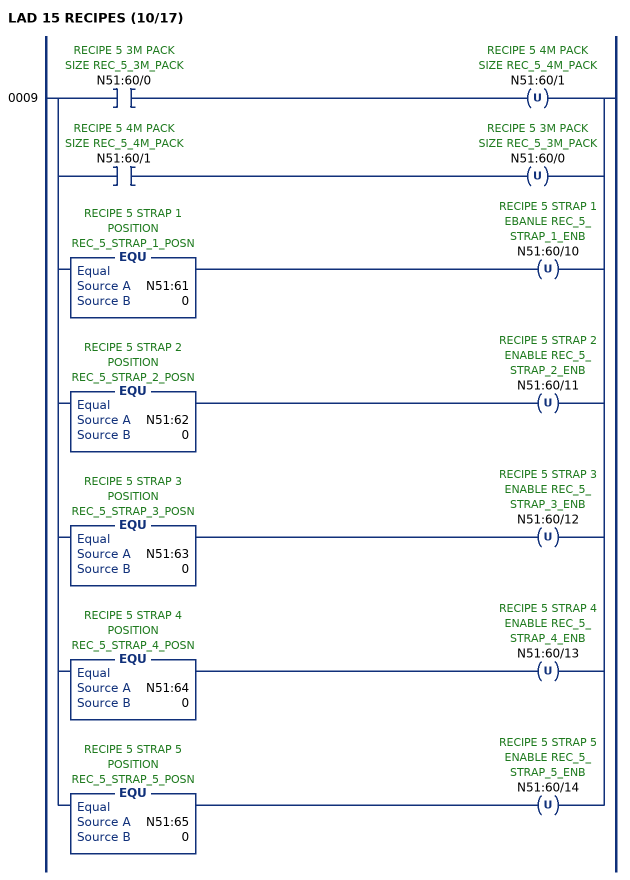
% Rung: 9 %
SOR BST XIC N51:60/0 OTU N51:60/1 NXB XIC N51:60/1 OTU N51:60/0 NXB EQU N51:61 0 OTU N51:60/10 NXB EQU N51:62 0 OTU N51:60/11 NXB EQU N51:63 0 OTU N51:60/12 NXB EQU N51:64 0 OTU N51:60/13 NXB EQU N51:65 0 OTU N51:60/14 BND EOR
%   N51:60/0  REC_5_3M_PACK  "RECIPE 5 3M PACK SIZE" %
%   N51:60/1  REC_5_4M_PACK  "RECIPE 5 4M PACK SIZE" %
%   N51:61  REC_5_STRAP_1_POSN  "RECIPE 5 STRAP 1 POSITION" %
%   N51:60/10  REC_5_STRAP_1_ENB  "RECIPE 5 STRAP 1 EBANLE" %
%   N51:62  REC_5_STRAP_2_POSN  "RECIPE 5 STRAP 2 POSITION" %
%   N51:60/11  REC_5_STRAP_2_ENB  "RECIPE 5 STRAP 2 ENABLE" %
%   N51:63  REC_5_STRAP_3_POSN  "RECIPE 5 STRAP 3 POSITION" %
%   N51:60/12  REC_5_STRAP_3_ENB  "RECIPE 5 STRAP 3 ENABLE" %
%   N51:64  REC_5_STRAP_4_POSN  "RECIPE 5 STRAP 4 POSITION" %
%   N51:60/13  REC_5_STRAP_4_ENB  "RECIPE 5 STRAP 4 ENABLE" %
%   N51:65  REC_5_STRAP_5_POSN  "RECIPE 5 STRAP 5 POSITION" %
%   N51:60/14  REC_5_STRAP_5_ENB  "RECIPE 5 STRAP 5 ENABLE" %

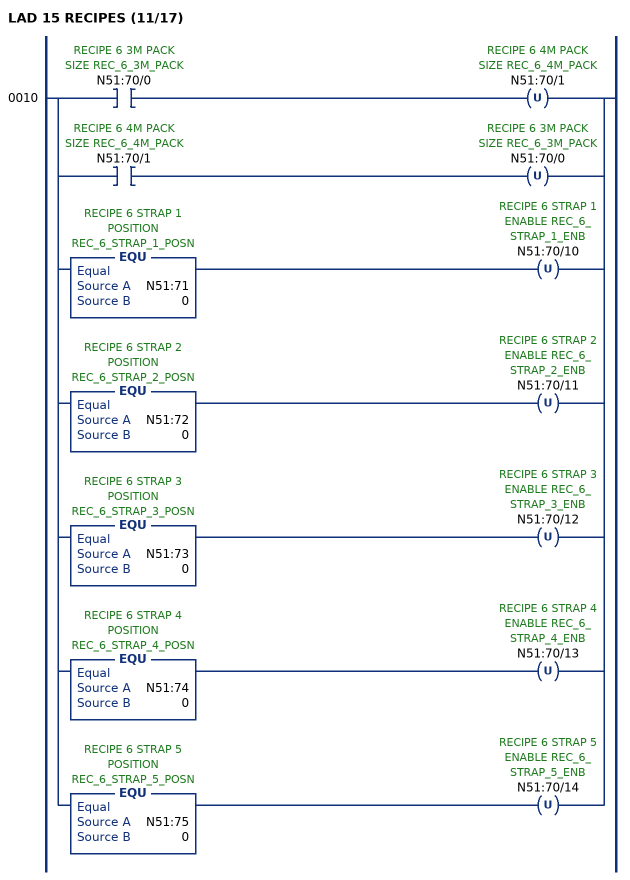
% Rung: 10 %
SOR BST XIC N51:70/0 OTU N51:70/1 NXB XIC N51:70/1 OTU N51:70/0 NXB EQU N51:71 0 OTU N51:70/10 NXB EQU N51:72 0 OTU N51:70/11 NXB EQU N51:73 0 OTU N51:70/12 NXB EQU N51:74 0 OTU N51:70/13 NXB EQU N51:75 0 OTU N51:70/14 BND EOR
%   N51:70/0  REC_6_3M_PACK  "RECIPE 6 3M PACK SIZE" %
%   N51:70/1  REC_6_4M_PACK  "RECIPE 6 4M PACK SIZE" %
%   N51:71  REC_6_STRAP_1_POSN  "RECIPE 6 STRAP 1 POSITION" %
%   N51:70/10  REC_6_STRAP_1_ENB  "RECIPE 6 STRAP 1 ENABLE" %
%   N51:72  REC_6_STRAP_2_POSN  "RECIPE 6 STRAP 2 POSITION" %
%   N51:70/11  REC_6_STRAP_2_ENB  "RECIPE 6 STRAP 2 ENABLE" %
%   N51:73  REC_6_STRAP_3_POSN  "RECIPE 6 STRAP 3 POSITION" %
%   N51:70/12  REC_6_STRAP_3_ENB  "RECIPE 6 STRAP 3 ENABLE" %
%   N51:74  REC_6_STRAP_4_POSN  "RECIPE 6 STRAP 4 POSITION" %
%   N51:70/13  REC_6_STRAP_4_ENB  "RECIPE 6 STRAP 4 ENABLE" %
%   N51:75  REC_6_STRAP_5_POSN  "RECIPE 6 STRAP 5 POSITION" %
%   N51:70/14  REC_6_STRAP_5_ENB  "RECIPE 6 STRAP 5 ENABLE" %

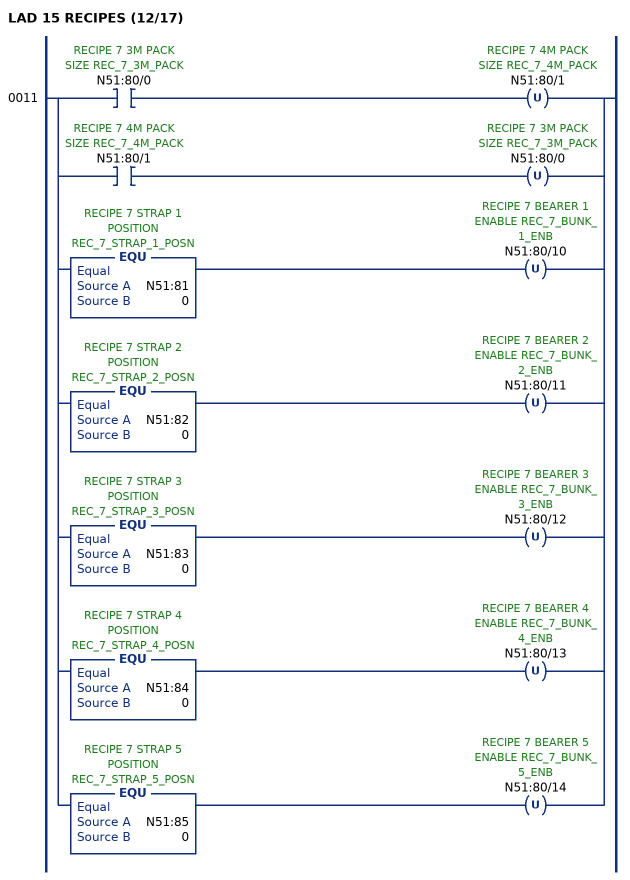
% Rung: 11 %
SOR BST XIC N51:80/0 OTU N51:80/1 NXB XIC N51:80/1 OTU N51:80/0 NXB EQU N51:81 0 OTU N51:80/10 NXB EQU N51:82 0 OTU N51:80/11 NXB EQU N51:83 0 OTU N51:80/12 NXB EQU N51:84 0 OTU N51:80/13 NXB EQU N51:85 0 OTU N51:80/14 BND EOR
%   N51:80/0  REC_7_3M_PACK  "RECIPE 7 3M PACK SIZE" %
%   N51:80/1  REC_7_4M_PACK  "RECIPE 7 4M PACK SIZE" %
%   N51:81  REC_7_STRAP_1_POSN  "RECIPE 7 STRAP 1 POSITION" %
%   N51:80/10  REC_7_BUNK_1_ENB  "RECIPE 7 BEARER 1 ENABLE" %
%   N51:82  REC_7_STRAP_2_POSN  "RECIPE 7 STRAP 2 POSITION" %
%   N51:80/11  REC_7_BUNK_2_ENB  "RECIPE 7 BEARER 2 ENABLE" %
%   N51:83  REC_7_STRAP_3_POSN  "RECIPE 7 STRAP 3 POSITION" %
%   N51:80/12  REC_7_BUNK_3_ENB  "RECIPE 7 BEARER 3 ENABLE" %
%   N51:84  REC_7_STRAP_4_POSN  "RECIPE 7 STRAP 4 POSITION" %
%   N51:80/13  REC_7_BUNK_4_ENB  "RECIPE 7 BEARER 4 ENABLE" %
%   N51:85  REC_7_STRAP_5_POSN  "RECIPE 7 STRAP 5 POSITION" %
%   N51:80/14  REC_7_BUNK_5_ENB  "RECIPE 7 BEARER 5 ENABLE" %

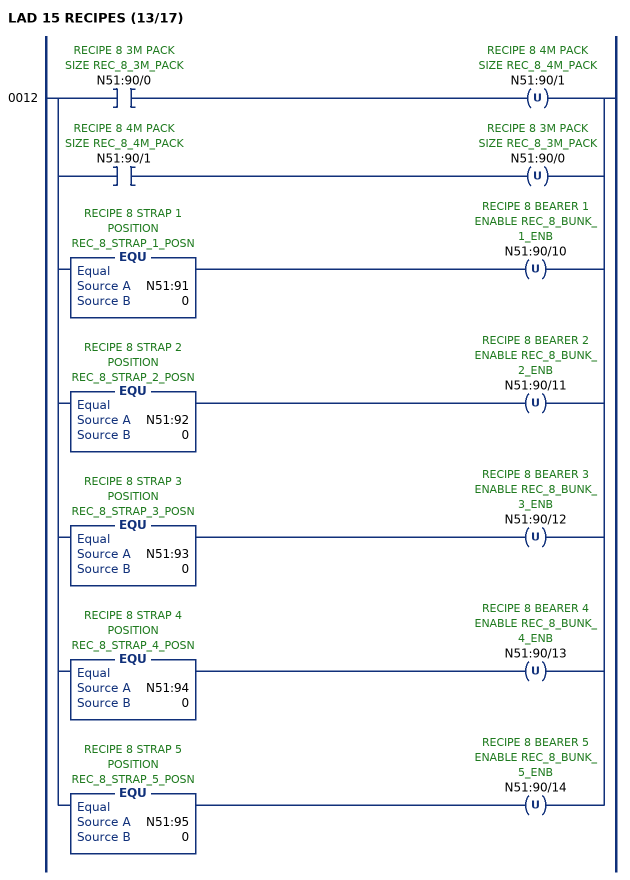
% Rung: 12 %
SOR BST XIC N51:90/0 OTU N51:90/1 NXB XIC N51:90/1 OTU N51:90/0 NXB EQU N51:91 0 OTU N51:90/10 NXB EQU N51:92 0 OTU N51:90/11 NXB EQU N51:93 0 OTU N51:90/12 NXB EQU N51:94 0 OTU N51:90/13 NXB EQU N51:95 0 OTU N51:90/14 BND EOR
%   N51:90/0  REC_8_3M_PACK  "RECIPE 8 3M PACK SIZE" %
%   N51:90/1  REC_8_4M_PACK  "RECIPE 8 4M PACK SIZE" %
%   N51:91  REC_8_STRAP_1_POSN  "RECIPE 8 STRAP 1 POSITION" %
%   N51:90/10  REC_8_BUNK_1_ENB  "RECIPE 8 BEARER 1 ENABLE" %
%   N51:92  REC_8_STRAP_2_POSN  "RECIPE 8 STRAP 2 POSITION" %
%   N51:90/11  REC_8_BUNK_2_ENB  "RECIPE 8 BEARER 2 ENABLE" %
%   N51:93  REC_8_STRAP_3_POSN  "RECIPE 8 STRAP 3 POSITION" %
%   N51:90/12  REC_8_BUNK_3_ENB  "RECIPE 8 BEARER 3 ENABLE" %
%   N51:94  REC_8_STRAP_4_POSN  "RECIPE 8 STRAP 4 POSITION" %
%   N51:90/13  REC_8_BUNK_4_ENB  "RECIPE 8 BEARER 4 ENABLE" %
%   N51:95  REC_8_STRAP_5_POSN  "RECIPE 8 STRAP 5 POSITION" %
%   N51:90/14  REC_8_BUNK_5_ENB  "RECIPE 8 BEARER 5 ENABLE" %

